FUNCTION_BLOCK FB_SaMElementManual EXTENDS FB_SaMElement
VAR
END_VAR

END_FUNCTION_BLOCK

(* stored: Version 1.1.0.1
   POU FB_SaMElementManual: Id {54e27e12-3d3f-0f17-3788-9da4dcb3548e}, SpecialFunc None *)
